TYPE checkDelayTime :
STRUCT
	//motor encoder and joint encoder deviation delay time
	Ti_armJntEncErr:TIME:=T#0.1S;
	//drive error delay time
	Ti_driveErr:TIME:=T#0.2S;
	//joint encoder ununuited delay time
	Ti_linkEncErr:TIME:=T#5S;
	Ti_linkEncErrCode:TIME:=T#10MS;
	//joint status error delay time 
	Ti_jntStatusErr:TIME:=T#1S;
	//spring breakage check time
	Ti_springBreakCheck:TIME:=T#0.3S;
	//motor hall check 
	Ti_motorHallCheck : TIME:=T#10MS;
	//motor phase check
	Ti_motorPhaseCheck : TIME:=T#10MS;
	//motor drive check
	Ti_motorDriveCheck : TIME:=T#10MS;
	//joint postion out of limit
	Ti_outOfLimit:TIME:=T#0.25S;
	//joint follow error delay time
	Ti_armJntFollowErr:TIME:=T#0.002S;
	//joint vel error delay time
	Ti_jntVelErr:TIME:=T#0.05S;
	//joint current error  delay time
	Ti_jntCurrentErr:TIME:=T#3S;
	//fixed point postion change of  master-slave state 
	Ti_fixedPointErr:TIME:=T#0.1S;
	//space pose error  delay time
	Ti_spacePoseErr:TIME:=T#0.002S;
	//commend joint position saltation delay time
	Ti_jntCmdSaltationErr:TIME:=T#0.002S;
	Ti_simCmdSaltaErr:TIME:=T#0.002S;
	//Deviation between command current and feedback current
	Ti_jntCmdCurrentErr:TIME:=T#0.5S;

	
	Ti_CarDualEncDev:TIME:=T#0.02S;
	Ti_CarDriveErr:TIME:=T#1S;
	Ti_CarActSec:TIME:=T#5S;
	Ti_CarActSecCode:TIME:=T#10mS;
	Ti_CarJntStatus:TIME:=T#1S;
	Ti_CarTorMotor:TIME:=T#20S;
	Ti_CaroutofLimit:TIME:=T#0.1S;
	Ti_CarFollowDev:TIME:=T#0.02S;
	Ti_CarJntVel:TIME:=T#0.05S;
	Ti_CarJntCurrent:TIME:=T#1S;
	Ti_CarMZDriveErr:TIME:=T#1S;
END_STRUCT
END_TYPE

(* stored: Version 1.1.0.1, ProductVersion 3.1.4024.11
   DUT checkDelayTime: Id {1842a9f8-6be9-44f3-b29d-ddeaee55cb3b} *)
